TYPE ST_BhFMControl :
STRUCT
	xReset	:	BOOL;
END_STRUCT
END_TYPE

(* stored: Version 1.1.0.1, ProductVersion 3.1.4020.12
   DUT ST_BhFMControl: Id {a8e6e27e-693a-4737-856d-d74c4803e4a7} *)
